{attribute 'linkalways'} 
{attribute 'no_explicit_call' := 'This FB is a CLASS and must be accessed using methods or properties'}
{attribute 'enable_dynamic_creation'}
FUNCTION_BLOCK FINAL GT_ULINT EXTENDS Node
VAR
	in1 : _ULINT(0);
	in2 : _ULINT(0);
	out : _BOOL(FALSE);
END_VAR

METHOD PUBLIC Clone : I_Node
VAR
	pNode : POINTER TO GT_ULINT;
END_VAR
pNode := __NEW(GT_ULINT);
Clone := pNode^;
END_METHOD

METHOD FB_init : BOOL
VAR_INPUT
	bInitRetains : BOOL; // if TRUE, the retain variables are initialized (warm start / cold start)
	bInCopyCode : BOOL;  // if TRUE, the instance afterwards gets moved into the copy code (online change)
END_VAR
AddInput('in1',THIS^.in1);
AddInput('in2',THIS^.in2);
AddOutput('out', THIS^.out);
END_METHOD

METHOD PROTECTED OnExecute
VAR
END_VAR
out.Value := in1.Value > in2.Value;
END_METHOD

END_FUNCTION_BLOCK

(* stored: Version 1.1.0.1, ProductVersion 3.1.4024.15
   POU GT_ULINT: Id {accb728f-8b44-40c8-ac56-194c2124702a}, SpecialFunc None
   Folder Constructor: Id {1f487cba-0be3-4ced-a85e-042b205a6547}
   Method Clone: Id {6cb54b5a-ff52-404c-b316-a4da6027c9b4}
   Method FB_init: Id {93220330-49af-4706-bbf4-8dfff3b90ced}
   Method OnExecute: Id {438e698a-2be3-4cf4-8537-61873b275220} *)
